// Mitsubishi GX Works2 project: LGCRFNW 23-01-2023_fr   PLC: Q06UDV

PROGRAM 00  // #1 Part Alarm
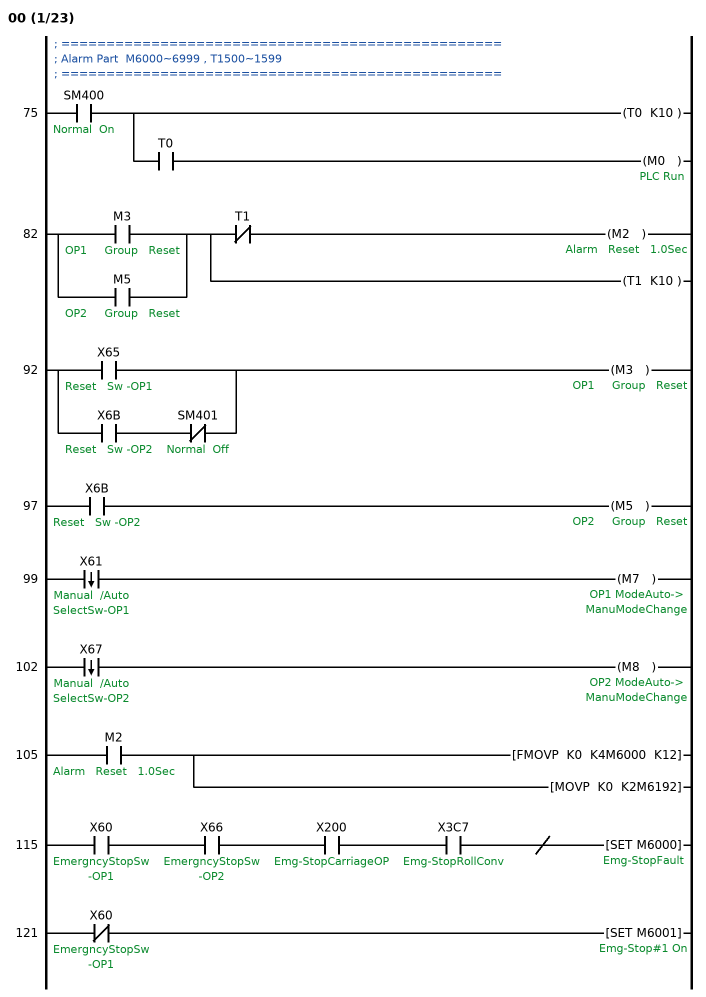
; =================================================
; Alarm Part  M6000~6999 , T1500~1599
; =================================================
75    LD      SM400  ; Normal  On
      OUT     T0 K10
      AND     T0
      OUT     M0  ; PLC Run
82    LD      M3  ; OP1     Group   Reset
      OR      M5  ; OP2     Group   Reset
      MPS
      ANI     T1
      OUT     M2  ; Alarm   Reset   1.0Sec
      MPP
      OUT     T1 K10
92    LD      X65  ; Reset   Sw -OP1
      LD      X6B  ; Reset   Sw -OP2
      ANI     SM401  ; Normal  Off
      ORB
      OUT     M3  ; OP1     Group   Reset
97    LD      X6B  ; Reset   Sw -OP2
      OUT     M5  ; OP2     Group   Reset
99    LDF     X61  ; Manual  /Auto   SelectSw-OP1
      OUT     M7  ; OP1 ModeAuto->  ManuModeChange
102   LDF     X67  ; Manual  /Auto   SelectSw-OP2
      OUT     M8  ; OP2 ModeAuto->  ManuModeChange
105   LD      M2  ; Alarm   Reset   1.0Sec
      FMOVP   K0 K4M6000 K12  ; Emg-StopFault
      MOVP    K0 K2M6192
115   LD      X60  ; EmergncyStopSw  -OP1
      AND     X66  ; EmergncyStopSw  -OP2
      AND     X200  ; Emg-StopCarriageOP
      AND     X3C7  ; Emg-StopRollConv
      INV
      SET     M6000  ; Emg-StopFault
121   LDI     X60  ; EmergncyStopSw  -OP1
      SET     M6001  ; Emg-Stop#1 On
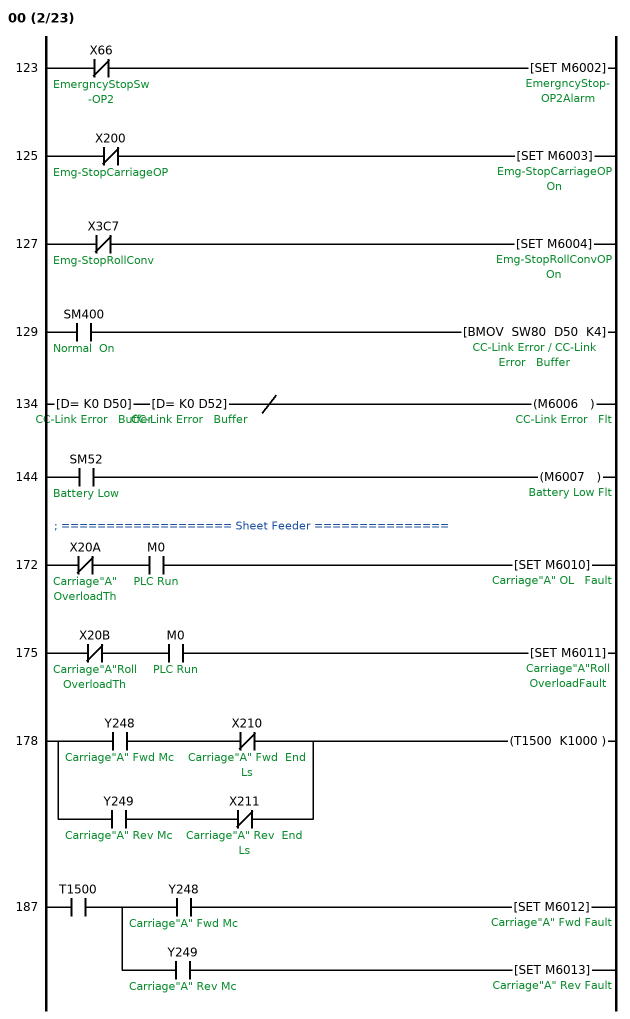
123   LDI     X66  ; EmergncyStopSw  -OP2
      SET     M6002  ; EmergncyStop-OP2Alarm
125   LDI     X200  ; Emg-StopCarriageOP
      SET     M6003  ; Emg-StopCarriageOP On
127   LDI     X3C7  ; Emg-StopRollConv
      SET     M6004  ; Emg-StopRollConvOP On
129   LD      SM400  ; Normal  On
      BMOV    SW80 D50 K4  ; CC-Link Error / CC-Link Error   Buffer
134   LDD=    K0 D50  ; CC-Link Error   Buffer
      ANDD=   K0 D52  ; CC-Link Error   Buffer
      INV
      OUT     M6006  ; CC-Link Error   Flt
144   LD      SM52  ; Battery Low
      OUT     M6007  ; Battery Low Flt
; =================== Sheet Feeder ===============
172   LDI     X20A  ; Carriage"A"     OverloadTh
      AND     M0  ; PLC Run
      SET     M6010  ; Carriage"A" OL   Fault
175   LDI     X20B  ; Carriage"A"Roll OverloadTh
      AND     M0  ; PLC Run
      SET     M6011  ; Carriage"A"Roll OverloadFault
178   LD      Y248  ; Carriage"A" Fwd Mc
      ANI     X210  ; Carriage"A" Fwd  End Ls
      LD      Y249  ; Carriage"A" Rev Mc
      ANI     X211  ; Carriage"A" Rev  End Ls
      ORB
      OUT     T1500 K1000
187   LD      T1500
      MPS
      AND     Y248  ; Carriage"A" Fwd Mc
      SET     M6012  ; Carriage"A" Fwd Fault
      MPP
      AND     Y249  ; Carriage"A" Rev Mc
      SET     M6013  ; Carriage"A" Rev Fault
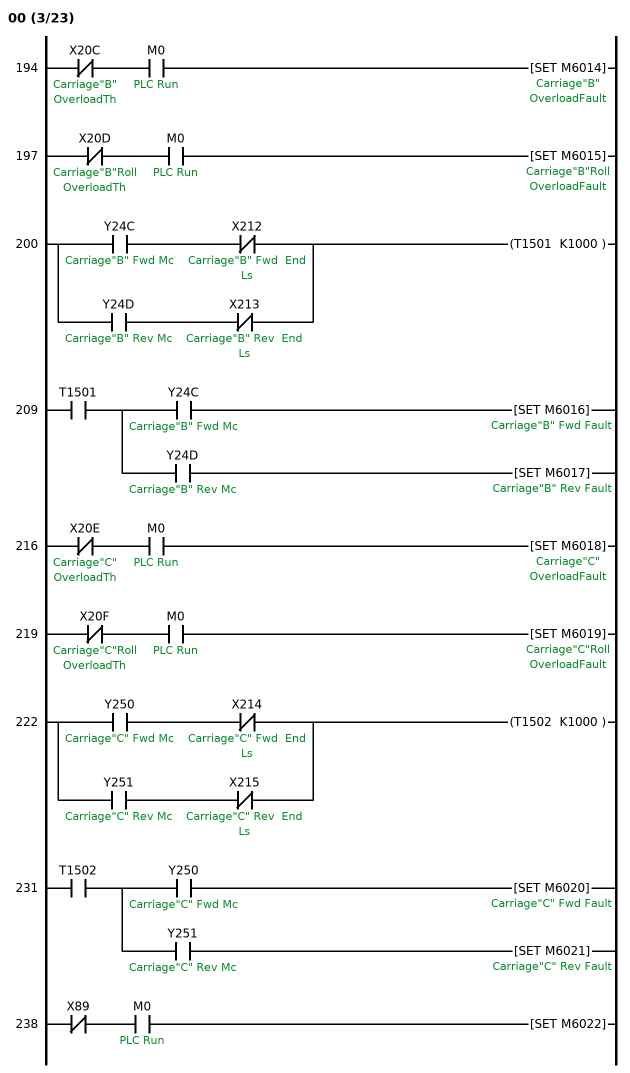
194   LDI     X20C  ; Carriage"B"     OverloadTh
      AND     M0  ; PLC Run
      SET     M6014  ; Carriage"B"     OverloadFault
197   LDI     X20D  ; Carriage"B"Roll OverloadTh
      AND     M0  ; PLC Run
      SET     M6015  ; Carriage"B"Roll OverloadFault
200   LD      Y24C  ; Carriage"B" Fwd Mc
      ANI     X212  ; Carriage"B" Fwd  End Ls
      LD      Y24D  ; Carriage"B" Rev Mc
      ANI     X213  ; Carriage"B" Rev  End Ls
      ORB
      OUT     T1501 K1000
209   LD      T1501
      MPS
      AND     Y24C  ; Carriage"B" Fwd Mc
      SET     M6016  ; Carriage"B" Fwd Fault
      MPP
      AND     Y24D  ; Carriage"B" Rev Mc
      SET     M6017  ; Carriage"B" Rev Fault
216   LDI     X20E  ; Carriage"C"     OverloadTh
      AND     M0  ; PLC Run
      SET     M6018  ; Carriage"C"     OverloadFault
219   LDI     X20F  ; Carriage"C"Roll OverloadTh
      AND     M0  ; PLC Run
      SET     M6019  ; Carriage"C"Roll OverloadFault
222   LD      Y250  ; Carriage"C" Fwd Mc
      ANI     X214  ; Carriage"C" Fwd  End Ls
      LD      Y251  ; Carriage"C" Rev Mc
      ANI     X215  ; Carriage"C" Rev  End Ls
      ORB
      OUT     T1502 K1000
231   LD      T1502
      MPS
      AND     Y250  ; Carriage"C" Fwd Mc
      SET     M6020  ; Carriage"C" Fwd Fault
      MPP
      AND     Y251  ; Carriage"C" Rev Mc
      SET     M6021  ; Carriage"C" Rev Fault
238   LDI     X89
      AND     M0  ; PLC Run
      SET     M6022
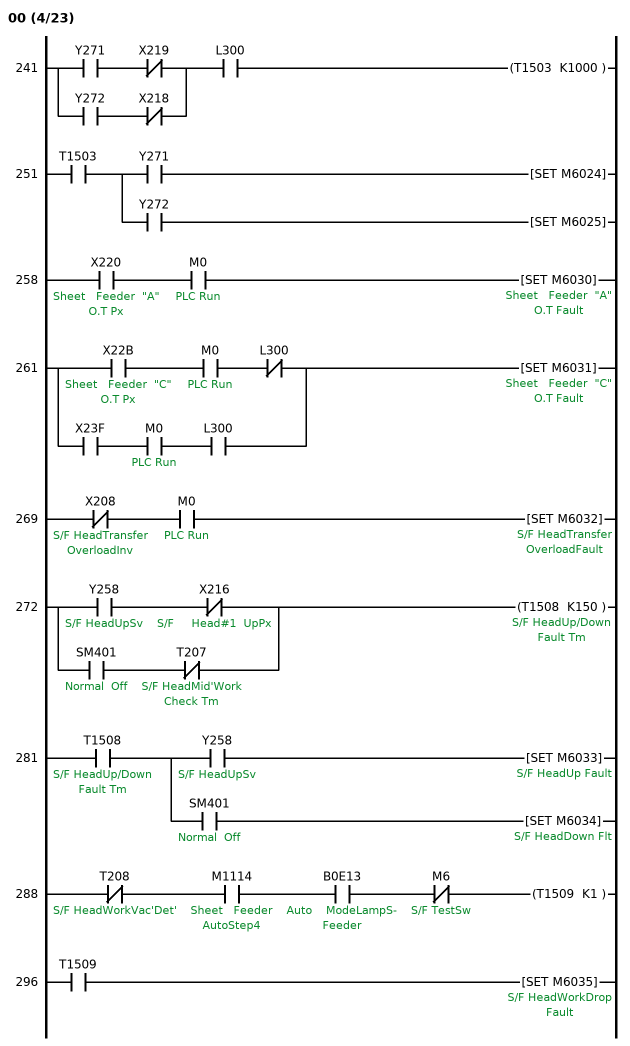
241   LD      Y271
      ANI     X219
      LD      Y272
      ANI     X218
      ORB
      AND     L300
      OUT     T1503 K1000
251   LD      T1503
      MPS
      AND     Y271
      SET     M6024
      MPP
      AND     Y272
      SET     M6025
258   LD      X220  ; Sheet   Feeder  "A" O.T Px
      AND     M0  ; PLC Run
      SET     M6030  ; Sheet   Feeder  "A" O.T Fault
261   LD      X22B  ; Sheet   Feeder  "C" O.T Px
      AND     M0  ; PLC Run
      ANI     L300
      LD      X23F
      AND     M0  ; PLC Run
      AND     L300
      ORB
      SET     M6031  ; Sheet   Feeder  "C" O.T Fault
269   LDI     X208  ; S/F HeadTransferOverloadInv
      AND     M0  ; PLC Run
      SET     M6032  ; S/F HeadTransferOverloadFault
272   LD      Y258  ; S/F HeadUpSv
      ANI     X216  ; S/F     Head#1  UpPx
      LD      SM401  ; Normal  Off
      ANI     T207  ; S/F HeadMid'WorkCheck Tm
      ORB
      OUT     T1508 K150  ; S/F HeadUp/Down Fault Tm
281   LD      T1508  ; S/F HeadUp/Down Fault Tm
      MPS
      AND     Y258  ; S/F HeadUpSv
      SET     M6033  ; S/F HeadUp Fault
      MPP
      AND     SM401  ; Normal  Off
      SET     M6034  ; S/F HeadDown Flt
288   LDI     T208  ; S/F HeadWorkVac'Det'
      AND     M1114  ; Sheet   Feeder  AutoStep4
      AND     B0E13  ; Auto    ModeLampS-Feeder
      ANI     M6  ; S/F TestSw
      OUT     T1509 K1
296   LD      T1509
      SET     M6035  ; S/F HeadWorkDropFault
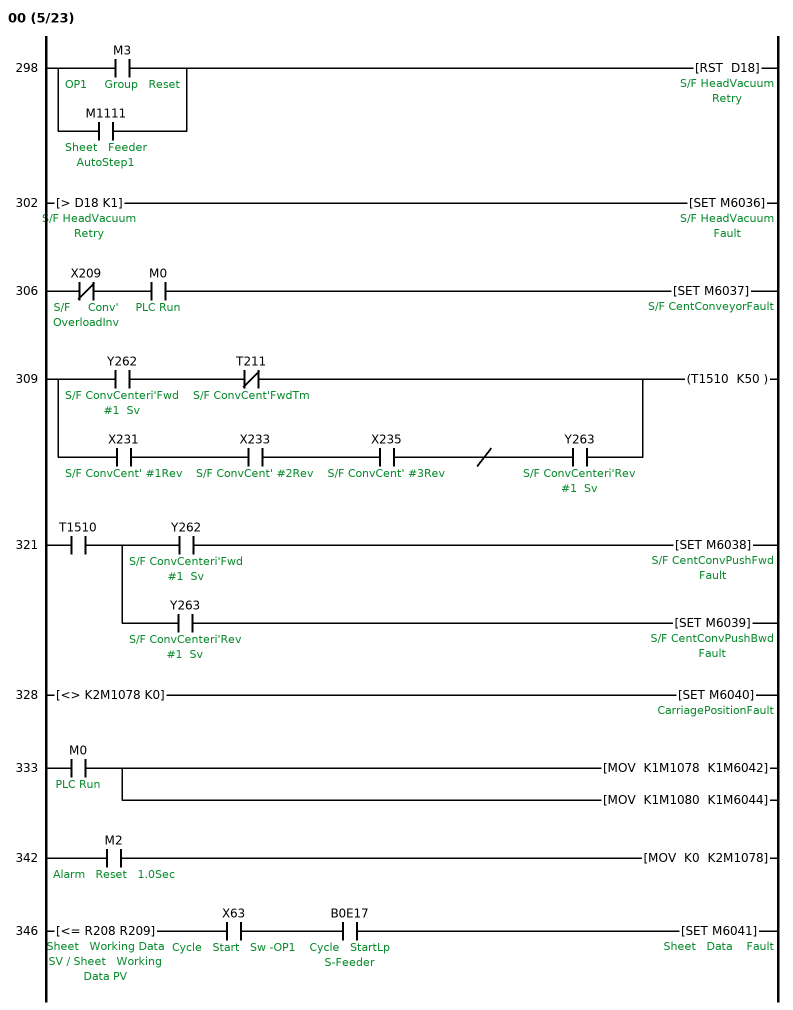
298   LD      M3  ; OP1     Group   Reset
      OR      M1111  ; Sheet   Feeder  AutoStep1
      RST     D18  ; S/F HeadVacuum  Retry
302   LD>     D18 K1  ; S/F HeadVacuum  Retry
      SET     M6036  ; S/F HeadVacuum  Fault
306   LDI     X209  ; S/F     Conv'   OverloadInv
      AND     M0  ; PLC Run
      SET     M6037  ; S/F CentConveyorFault
309   LD      Y262  ; S/F ConvCenteri'Fwd #1  Sv
      ANI     T211  ; S/F ConvCent'FwdTm
      LD      X231  ; S/F ConvCent' #1Rev
      AND     X233  ; S/F ConvCent' #2Rev
      AND     X235  ; S/F ConvCent' #3Rev
      INV
      AND     Y263  ; S/F ConvCenteri'Rev #1  Sv
      ORB
      OUT     T1510 K50
321   LD      T1510
      MPS
      AND     Y262  ; S/F ConvCenteri'Fwd #1  Sv
      SET     M6038  ; S/F CentConvPushFwdFault
      MPP
      AND     Y263  ; S/F ConvCenteri'Rev #1  Sv
      SET     M6039  ; S/F CentConvPushBwdFault
328   LD<>    K2M1078 K0  ; Carriage#1 Pos' Fault
      SET     M6040  ; CarriagePositionFault
333   LD      M0  ; PLC Run
      MOV     K1M1078 K1M6042
      MOV     K1M1080 K1M6044  ; Carriage#3 Pos'  Fault
342   LD      M2  ; Alarm   Reset   1.0Sec
      MOV     K0 K2M1078
346   LD<=    R208 R209  ; Sheet   Working Data SV / Sheet   Working Data PV
      AND     X63  ; Cycle   Start   Sw -OP1
      AND     B0E17  ; Cycle   StartLp S-Feeder
      SET     M6041  ; Sheet   Data    Fault
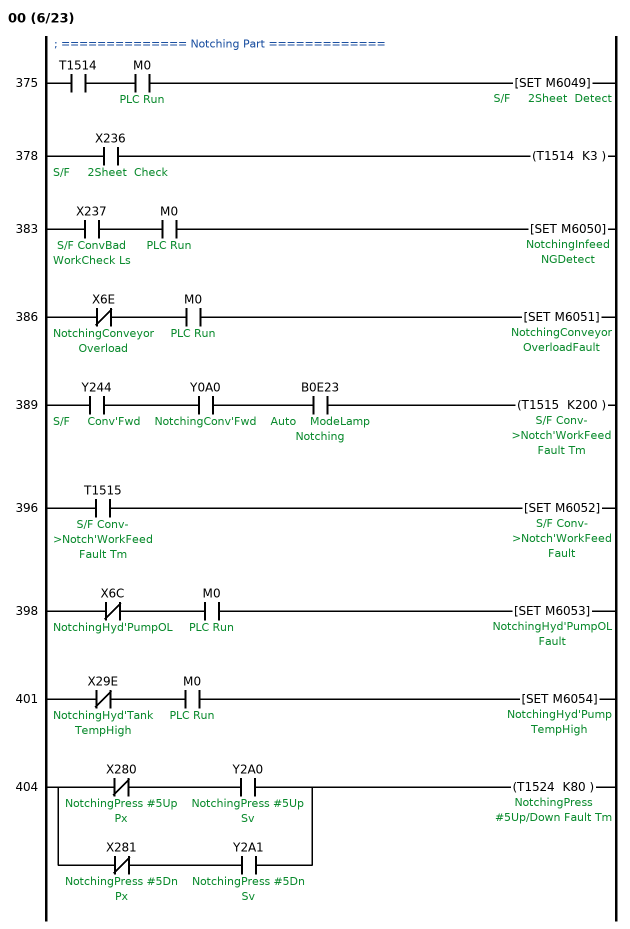
; ============== Notching Part =============
375   LD      T1514
      AND     M0  ; PLC Run
      SET     M6049  ; S/F     2Sheet  Detect
378   LD      X236  ; S/F     2Sheet  Check
      OUT     T1514 K3
383   LD      X237  ; S/F ConvBad WorkCheck Ls
      AND     M0  ; PLC Run
      SET     M6050  ; NotchingInfeedNGDetect
386   LDI     X6E  ; NotchingConveyorOverload
      AND     M0  ; PLC Run
      SET     M6051  ; NotchingConveyorOverloadFault
389   LD      Y244  ; S/F     Conv'Fwd
      AND     Y0A0  ; NotchingConv'Fwd
      AND     B0E23  ; Auto    ModeLampNotching
      OUT     T1515 K200  ; S/F Conv->Notch'WorkFeedFault Tm
396   LD      T1515  ; S/F Conv->Notch'WorkFeedFault Tm
      SET     M6052  ; S/F Conv->Notch'WorkFeedFault
398   LDI     X6C  ; NotchingHyd'PumpOL
      AND     M0  ; PLC Run
      SET     M6053  ; NotchingHyd'PumpOL Fault
401   LDI     X29E  ; NotchingHyd'TankTempHigh
      AND     M0  ; PLC Run
      SET     M6054  ; NotchingHyd'PumpTempHigh
404   LDI     X280  ; NotchingPress #5Up Px
      AND     Y2A0  ; NotchingPress #5Up Sv
      LDI     X281  ; NotchingPress #5Dn Px
      AND     Y2A1  ; NotchingPress #5Dn Sv
      ORB
      OUT     T1524 K80  ; NotchingPress #5Up/Down Fault Tm
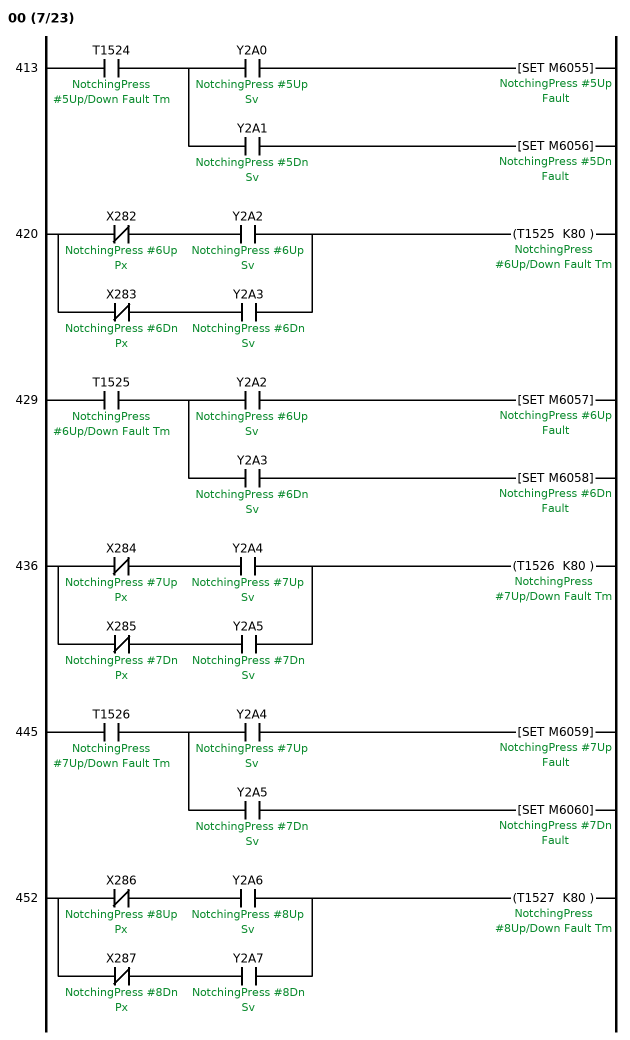
413   LD      T1524  ; NotchingPress #5Up/Down Fault Tm
      MPS
      AND     Y2A0  ; NotchingPress #5Up Sv
      SET     M6055  ; NotchingPress #5Up Fault
      MPP
      AND     Y2A1  ; NotchingPress #5Dn Sv
      SET     M6056  ; NotchingPress #5Dn Fault
420   LDI     X282  ; NotchingPress #6Up Px
      AND     Y2A2  ; NotchingPress #6Up Sv
      LDI     X283  ; NotchingPress #6Dn Px
      AND     Y2A3  ; NotchingPress #6Dn Sv
      ORB
      OUT     T1525 K80  ; NotchingPress #6Up/Down Fault Tm
429   LD      T1525  ; NotchingPress #6Up/Down Fault Tm
      MPS
      AND     Y2A2  ; NotchingPress #6Up Sv
      SET     M6057  ; NotchingPress #6Up Fault
      MPP
      AND     Y2A3  ; NotchingPress #6Dn Sv
      SET     M6058  ; NotchingPress #6Dn Fault
436   LDI     X284  ; NotchingPress #7Up Px
      AND     Y2A4  ; NotchingPress #7Up Sv
      LDI     X285  ; NotchingPress #7Dn Px
      AND     Y2A5  ; NotchingPress #7Dn Sv
      ORB
      OUT     T1526 K80  ; NotchingPress #7Up/Down Fault Tm
445   LD      T1526  ; NotchingPress #7Up/Down Fault Tm
      MPS
      AND     Y2A4  ; NotchingPress #7Up Sv
      SET     M6059  ; NotchingPress #7Up Fault
      MPP
      AND     Y2A5  ; NotchingPress #7Dn Sv
      SET     M6060  ; NotchingPress #7Dn Fault
452   LDI     X286  ; NotchingPress #8Up Px
      AND     Y2A6  ; NotchingPress #8Up Sv
      LDI     X287  ; NotchingPress #8Dn Px
      AND     Y2A7  ; NotchingPress #8Dn Sv
      ORB
      OUT     T1527 K80  ; NotchingPress #8Up/Down Fault Tm
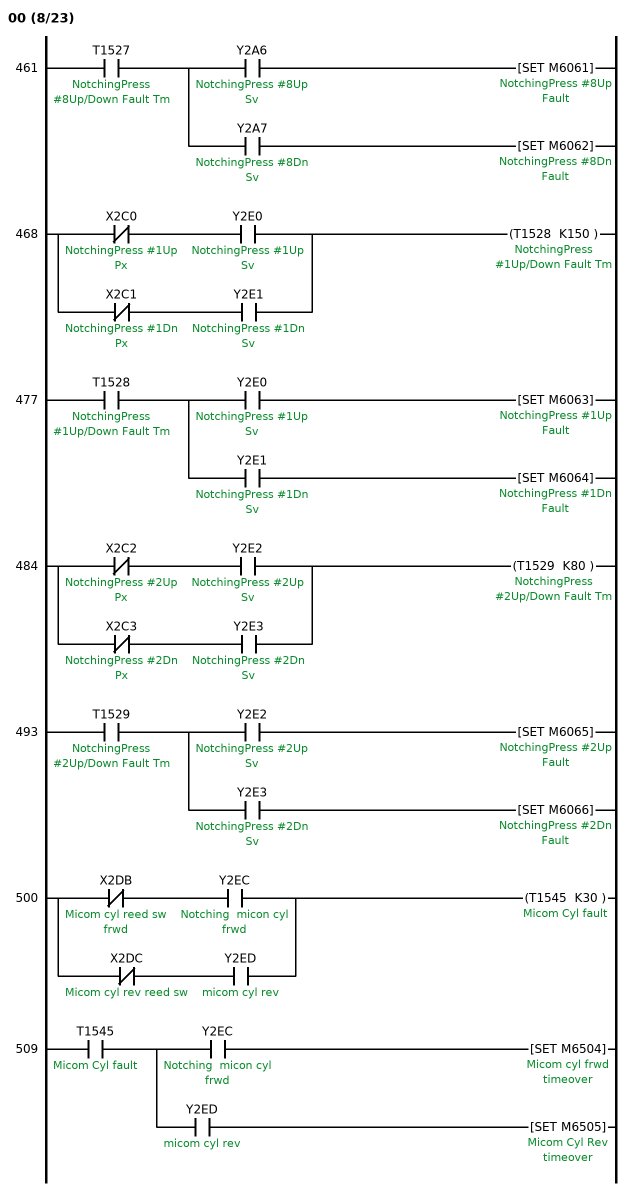
461   LD      T1527  ; NotchingPress #8Up/Down Fault Tm
      MPS
      AND     Y2A6  ; NotchingPress #8Up Sv
      SET     M6061  ; NotchingPress #8Up Fault
      MPP
      AND     Y2A7  ; NotchingPress #8Dn Sv
      SET     M6062  ; NotchingPress #8Dn Fault
468   LDI     X2C0  ; NotchingPress #1Up Px
      AND     Y2E0  ; NotchingPress #1Up Sv
      LDI     X2C1  ; NotchingPress #1Dn Px
      AND     Y2E1  ; NotchingPress #1Dn Sv
      ORB
      OUT     T1528 K150  ; NotchingPress #1Up/Down Fault Tm
477   LD      T1528  ; NotchingPress #1Up/Down Fault Tm
      MPS
      AND     Y2E0  ; NotchingPress #1Up Sv
      SET     M6063  ; NotchingPress #1Up Fault
      MPP
      AND     Y2E1  ; NotchingPress #1Dn Sv
      SET     M6064  ; NotchingPress #1Dn Fault
484   LDI     X2C2  ; NotchingPress #2Up Px
      AND     Y2E2  ; NotchingPress #2Up Sv
      LDI     X2C3  ; NotchingPress #2Dn Px
      AND     Y2E3  ; NotchingPress #2Dn Sv
      ORB
      OUT     T1529 K80  ; NotchingPress #2Up/Down Fault Tm
493   LD      T1529  ; NotchingPress #2Up/Down Fault Tm
      MPS
      AND     Y2E2  ; NotchingPress #2Up Sv
      SET     M6065  ; NotchingPress #2Up Fault
      MPP
      AND     Y2E3  ; NotchingPress #2Dn Sv
      SET     M6066  ; NotchingPress #2Dn Fault
500   LDI     X2DB  ; Micom cyl reed sw frwd
      AND     Y2EC  ; Notching  micon cyl frwd
      LDI     X2DC  ; Micom cyl rev reed sw
      AND     Y2ED  ; micom cyl rev
      ORB
      OUT     T1545 K30  ; Micom Cyl fault
509   LD      T1545  ; Micom Cyl fault
      MPS
      AND     Y2EC  ; Notching  micon cyl frwd
      SET     M6504  ; Micom cyl frwd timeover
      MPP
      AND     Y2ED  ; micom cyl rev
      SET     M6505  ; Micom Cyl Rev timeover
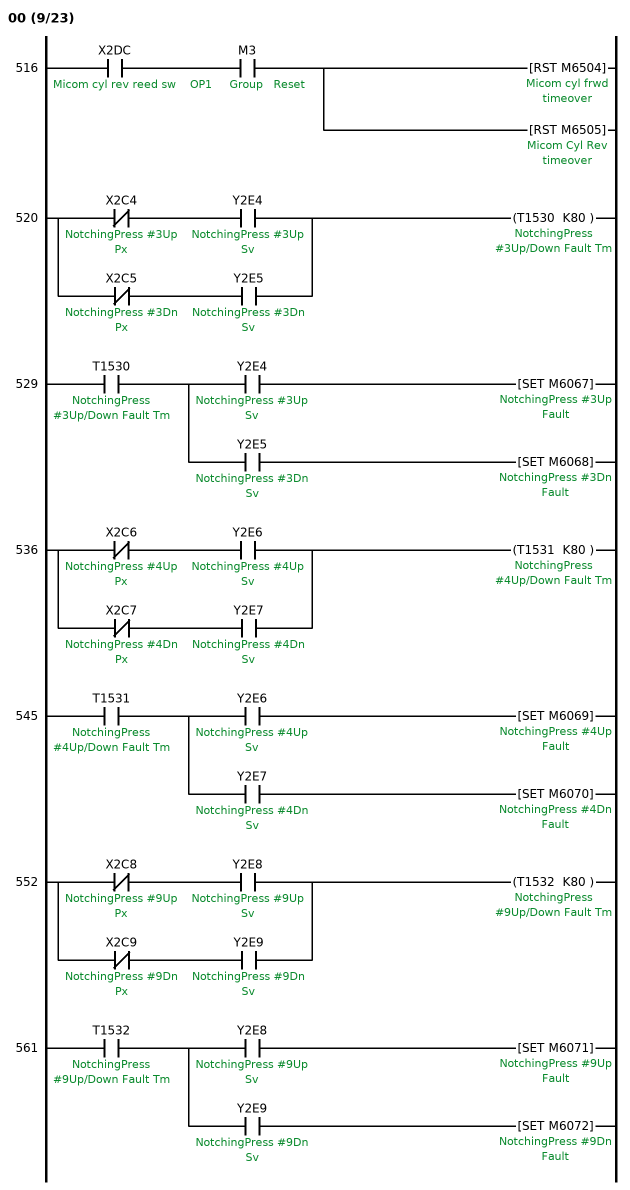
516   LD      X2DC  ; Micom cyl rev reed sw
      AND     M3  ; OP1     Group   Reset
      RST     M6504  ; Micom cyl frwd timeover
      RST     M6505  ; Micom Cyl Rev timeover
520   LDI     X2C4  ; NotchingPress #3Up Px
      AND     Y2E4  ; NotchingPress #3Up Sv
      LDI     X2C5  ; NotchingPress #3Dn Px
      AND     Y2E5  ; NotchingPress #3Dn Sv
      ORB
      OUT     T1530 K80  ; NotchingPress #3Up/Down Fault Tm
529   LD      T1530  ; NotchingPress #3Up/Down Fault Tm
      MPS
      AND     Y2E4  ; NotchingPress #3Up Sv
      SET     M6067  ; NotchingPress #3Up Fault
      MPP
      AND     Y2E5  ; NotchingPress #3Dn Sv
      SET     M6068  ; NotchingPress #3Dn Fault
536   LDI     X2C6  ; NotchingPress #4Up Px
      AND     Y2E6  ; NotchingPress #4Up Sv
      LDI     X2C7  ; NotchingPress #4Dn Px
      AND     Y2E7  ; NotchingPress #4Dn Sv
      ORB
      OUT     T1531 K80  ; NotchingPress #4Up/Down Fault Tm
545   LD      T1531  ; NotchingPress #4Up/Down Fault Tm
      MPS
      AND     Y2E6  ; NotchingPress #4Up Sv
      SET     M6069  ; NotchingPress #4Up Fault
      MPP
      AND     Y2E7  ; NotchingPress #4Dn Sv
      SET     M6070  ; NotchingPress #4Dn Fault
552   LDI     X2C8  ; NotchingPress #9Up Px
      AND     Y2E8  ; NotchingPress #9Up Sv
      LDI     X2C9  ; NotchingPress #9Dn Px
      AND     Y2E9  ; NotchingPress #9Dn Sv
      ORB
      OUT     T1532 K80  ; NotchingPress #9Up/Down Fault Tm
561   LD      T1532  ; NotchingPress #9Up/Down Fault Tm
      MPS
      AND     Y2E8  ; NotchingPress #9Up Sv
      SET     M6071  ; NotchingPress #9Up Fault
      MPP
      AND     Y2E9  ; NotchingPress #9Dn Sv
      SET     M6072  ; NotchingPress #9Dn Fault
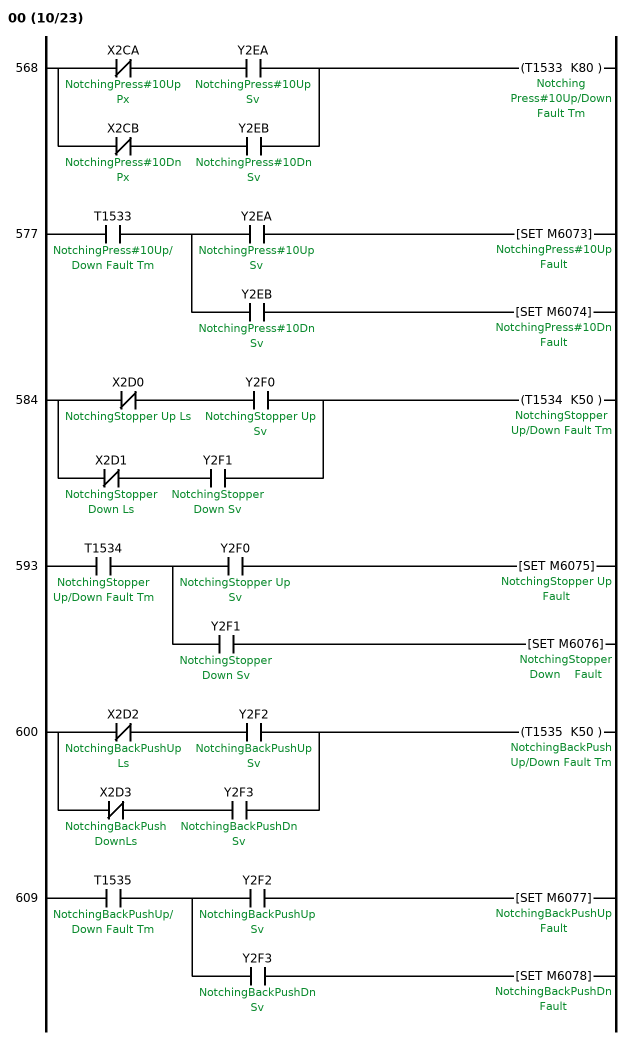
568   LDI     X2CA  ; NotchingPress#10Up Px
      AND     Y2EA  ; NotchingPress#10Up Sv
      LDI     X2CB  ; NotchingPress#10Dn Px
      AND     Y2EB  ; NotchingPress#10Dn Sv
      ORB
      OUT     T1533 K80  ; NotchingPress#10Up/Down Fault Tm
577   LD      T1533  ; NotchingPress#10Up/Down Fault Tm
      MPS
      AND     Y2EA  ; NotchingPress#10Up Sv
      SET     M6073  ; NotchingPress#10Up Fault
      MPP
      AND     Y2EB  ; NotchingPress#10Dn Sv
      SET     M6074  ; NotchingPress#10Dn Fault
584   LDI     X2D0  ; NotchingStopper Up Ls
      AND     Y2F0  ; NotchingStopper Up Sv
      LDI     X2D1  ; NotchingStopper Down Ls
      AND     Y2F1  ; NotchingStopper Down Sv
      ORB
      OUT     T1534 K50  ; NotchingStopper Up/Down Fault Tm
593   LD      T1534  ; NotchingStopper Up/Down Fault Tm
      MPS
      AND     Y2F0  ; NotchingStopper Up Sv
      SET     M6075  ; NotchingStopper Up Fault
      MPP
      AND     Y2F1  ; NotchingStopper Down Sv
      SET     M6076  ; NotchingStopper Down    Fault
600   LDI     X2D2  ; NotchingBackPushUpLs
      AND     Y2F2  ; NotchingBackPushUpSv
      LDI     X2D3  ; NotchingBackPushDownLs
      AND     Y2F3  ; NotchingBackPushDnSv
      ORB
      OUT     T1535 K50  ; NotchingBackPushUp/Down Fault Tm
609   LD      T1535  ; NotchingBackPushUp/Down Fault Tm
      MPS
      AND     Y2F2  ; NotchingBackPushUpSv
      SET     M6077  ; NotchingBackPushUpFault
      MPP
      AND     Y2F3  ; NotchingBackPushDnSv
      SET     M6078  ; NotchingBackPushDnFault
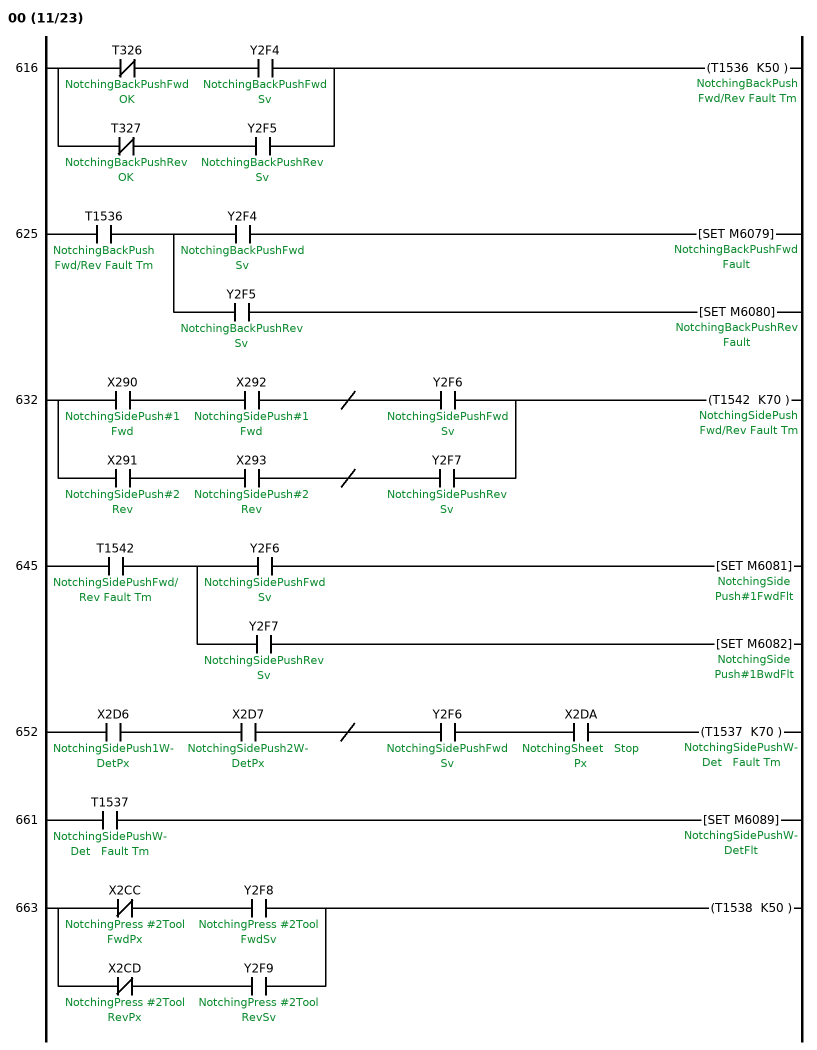
616   LDI     T326  ; NotchingBackPushFwd OK
      AND     Y2F4  ; NotchingBackPushFwdSv
      LDI     T327  ; NotchingBackPushRev OK
      AND     Y2F5  ; NotchingBackPushRevSv
      ORB
      OUT     T1536 K50  ; NotchingBackPushFwd/Rev Fault Tm
625   LD      T1536  ; NotchingBackPushFwd/Rev Fault Tm
      MPS
      AND     Y2F4  ; NotchingBackPushFwdSv
      SET     M6079  ; NotchingBackPushFwdFault
      MPP
      AND     Y2F5  ; NotchingBackPushRevSv
      SET     M6080  ; NotchingBackPushRevFault
632   LD      X290  ; NotchingSidePush#1 Fwd
      AND     X292  ; NotchingSidePush#1 Fwd
      INV
      AND     Y2F6  ; NotchingSidePushFwd Sv
      LD      X291  ; NotchingSidePush#2 Rev
      AND     X293  ; NotchingSidePush#2 Rev
      INV
      AND     Y2F7  ; NotchingSidePushRev Sv
      ORB
      OUT     T1542 K70  ; NotchingSidePushFwd/Rev Fault Tm
645   LD      T1542  ; NotchingSidePushFwd/Rev Fault Tm
      MPS
      AND     Y2F6  ; NotchingSidePushFwd Sv
      SET     M6081  ; NotchingSidePush#1FwdFlt
      MPP
      AND     Y2F7  ; NotchingSidePushRev Sv
      SET     M6082  ; NotchingSidePush#1BwdFlt
652   LD      X2D6  ; NotchingSidePush1W-DetPx
      AND     X2D7  ; NotchingSidePush2W-DetPx
      INV
      AND     Y2F6  ; NotchingSidePushFwd Sv
      AND     X2DA  ; NotchingSheet   Stop Px
      OUT     T1537 K70  ; NotchingSidePushW-Det   Fault Tm
661   LD      T1537  ; NotchingSidePushW-Det   Fault Tm
      SET     M6089  ; NotchingSidePushW-DetFlt
663   LDI     X2CC  ; NotchingPress #2Tool FwdPx
      AND     Y2F8  ; NotchingPress #2Tool FwdSv
      LDI     X2CD  ; NotchingPress #2Tool RevPx
      AND     Y2F9  ; NotchingPress #2Tool RevSv
      ORB
      OUT     T1538 K50
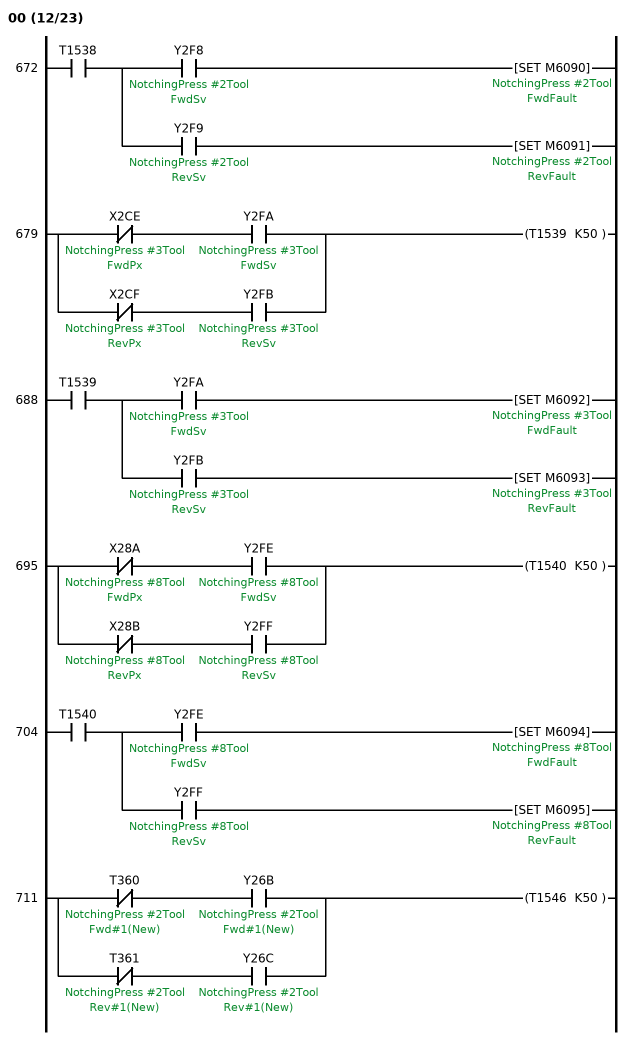
672   LD      T1538
      MPS
      AND     Y2F8  ; NotchingPress #2Tool FwdSv
      SET     M6090  ; NotchingPress #2Tool FwdFault
      MPP
      AND     Y2F9  ; NotchingPress #2Tool RevSv
      SET     M6091  ; NotchingPress #2Tool RevFault
679   LDI     X2CE  ; NotchingPress #3Tool FwdPx
      AND     Y2FA  ; NotchingPress #3Tool FwdSv
      LDI     X2CF  ; NotchingPress #3Tool RevPx
      AND     Y2FB  ; NotchingPress #3Tool RevSv
      ORB
      OUT     T1539 K50
688   LD      T1539
      MPS
      AND     Y2FA  ; NotchingPress #3Tool FwdSv
      SET     M6092  ; NotchingPress #3Tool FwdFault
      MPP
      AND     Y2FB  ; NotchingPress #3Tool RevSv
      SET     M6093  ; NotchingPress #3Tool RevFault
695   LDI     X28A  ; NotchingPress #8Tool FwdPx
      AND     Y2FE  ; NotchingPress #8Tool FwdSv
      LDI     X28B  ; NotchingPress #8Tool RevPx
      AND     Y2FF  ; NotchingPress #8Tool RevSv
      ORB
      OUT     T1540 K50
704   LD      T1540
      MPS
      AND     Y2FE  ; NotchingPress #8Tool FwdSv
      SET     M6094  ; NotchingPress #8Tool FwdFault
      MPP
      AND     Y2FF  ; NotchingPress #8Tool RevSv
      SET     M6095  ; NotchingPress #8Tool RevFault
711   LDI     T360  ; NotchingPress #2Tool Fwd#1(New)
      AND     Y26B  ; NotchingPress #2Tool Fwd#1(New)
      LDI     T361  ; NotchingPress #2Tool Rev#1(New)
      AND     Y26C  ; NotchingPress #2Tool Rev#1(New)
      ORB
      OUT     T1546 K50
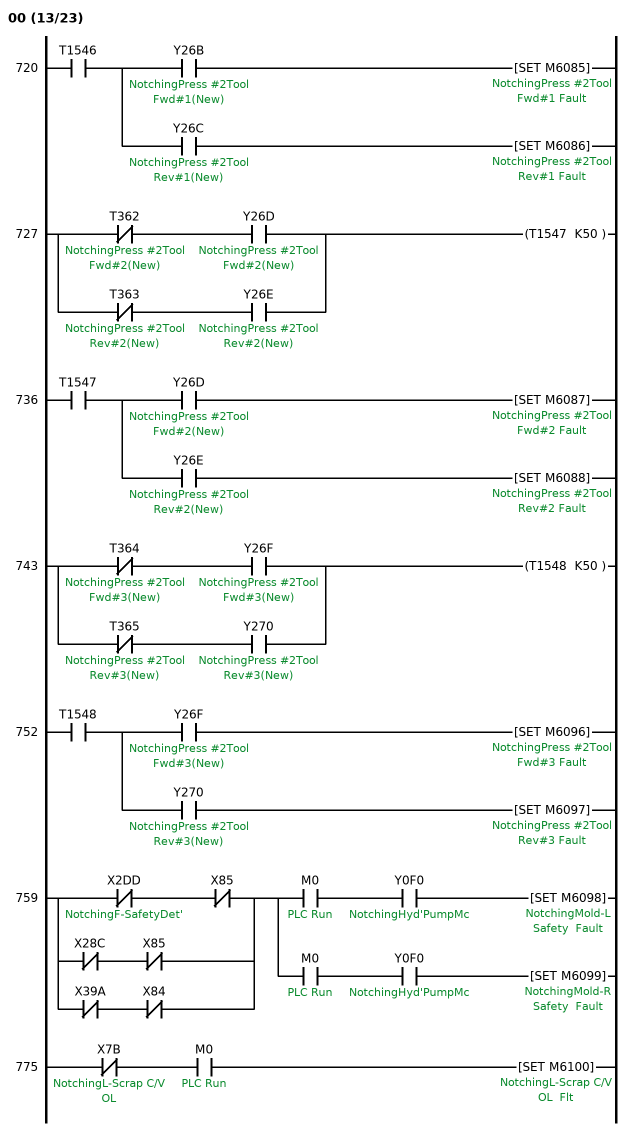
720   LD      T1546
      MPS
      AND     Y26B  ; NotchingPress #2Tool Fwd#1(New)
      SET     M6085  ; NotchingPress #2Tool Fwd#1 Fault
      MPP
      AND     Y26C  ; NotchingPress #2Tool Rev#1(New)
      SET     M6086  ; NotchingPress #2Tool Rev#1 Fault
727   LDI     T362  ; NotchingPress #2Tool Fwd#2(New)
      AND     Y26D  ; NotchingPress #2Tool Fwd#2(New)
      LDI     T363  ; NotchingPress #2Tool Rev#2(New)
      AND     Y26E  ; NotchingPress #2Tool Rev#2(New)
      ORB
      OUT     T1547 K50
736   LD      T1547
      MPS
      AND     Y26D  ; NotchingPress #2Tool Fwd#2(New)
      SET     M6087  ; NotchingPress #2Tool Fwd#2 Fault
      MPP
      AND     Y26E  ; NotchingPress #2Tool Rev#2(New)
      SET     M6088  ; NotchingPress #2Tool Rev#2 Fault
743   LDI     T364  ; NotchingPress #2Tool Fwd#3(New)
      AND     Y26F  ; NotchingPress #2Tool Fwd#3(New)
      LDI     T365  ; NotchingPress #2Tool Rev#3(New)
      AND     Y270  ; NotchingPress #2Tool Rev#3(New)
      ORB
      OUT     T1548 K50
752   LD      T1548
      MPS
      AND     Y26F  ; NotchingPress #2Tool Fwd#3(New)
      SET     M6096  ; NotchingPress #2Tool Fwd#3 Fault
      MPP
      AND     Y270  ; NotchingPress #2Tool Rev#3(New)
      SET     M6097  ; NotchingPress #2Tool Rev#3 Fault
759   LDI     X2DD  ; NotchingF-SafetyDet'
      ANI     X85
      LDI     X28C
      ANI     X85
      ORB
      LDI     X39A
      ANI     X84
      ORB
      MPS
      AND     M0  ; PLC Run
      AND     Y0F0  ; NotchingHyd'PumpMc
      SET     M6098  ; NotchingMold-L  Safety  Fault
      MPP
      AND     M0  ; PLC Run
      AND     Y0F0  ; NotchingHyd'PumpMc
      SET     M6099  ; NotchingMold-R  Safety  Fault
775   LDI     X7B  ; NotchingL-Scrap C/V OL
      AND     M0  ; PLC Run
      SET     M6100  ; NotchingL-Scrap C/V OL  Flt
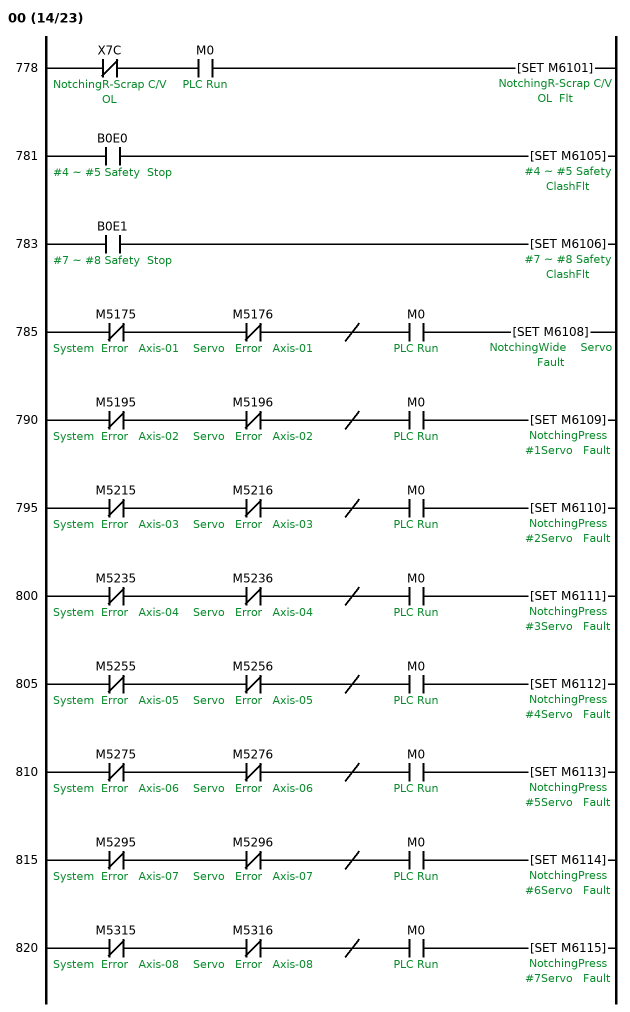
778   LDI     X7C  ; NotchingR-Scrap C/V OL
      AND     M0  ; PLC Run
      SET     M6101  ; NotchingR-Scrap C/V OL  Flt
781   LD      B0E0  ; #4 ~ #5 Safety  Stop
      SET     M6105  ; #4 ~ #5 Safety  ClashFlt
783   LD      B0E1  ; #7 ~ #8 Safety  Stop
      SET     M6106  ; #7 ~ #8 Safety  ClashFlt
785   LDI     M5175  ; System  Error   Axis-01
      ANI     M5176  ; Servo   Error   Axis-01
      INV
      AND     M0  ; PLC Run
      SET     M6108  ; NotchingWide    Servo   Fault
790   LDI     M5195  ; System  Error   Axis-02
      ANI     M5196  ; Servo   Error   Axis-02
      INV
      AND     M0  ; PLC Run
      SET     M6109  ; NotchingPress #1Servo   Fault
795   LDI     M5215  ; System  Error   Axis-03
      ANI     M5216  ; Servo   Error   Axis-03
      INV
      AND     M0  ; PLC Run
      SET     M6110  ; NotchingPress #2Servo   Fault
800   LDI     M5235  ; System  Error   Axis-04
      ANI     M5236  ; Servo   Error   Axis-04
      INV
      AND     M0  ; PLC Run
      SET     M6111  ; NotchingPress #3Servo   Fault
805   LDI     M5255  ; System  Error   Axis-05
      ANI     M5256  ; Servo   Error   Axis-05
      INV
      AND     M0  ; PLC Run
      SET     M6112  ; NotchingPress #4Servo   Fault
810   LDI     M5275  ; System  Error   Axis-06
      ANI     M5276  ; Servo   Error   Axis-06
      INV
      AND     M0  ; PLC Run
      SET     M6113  ; NotchingPress #5Servo   Fault
815   LDI     M5295  ; System  Error   Axis-07
      ANI     M5296  ; Servo   Error   Axis-07
      INV
      AND     M0  ; PLC Run
      SET     M6114  ; NotchingPress #6Servo   Fault
820   LDI     M5315  ; System  Error   Axis-08
      ANI     M5316  ; Servo   Error   Axis-08
      INV
      AND     M0  ; PLC Run
      SET     M6115  ; NotchingPress #7Servo   Fault
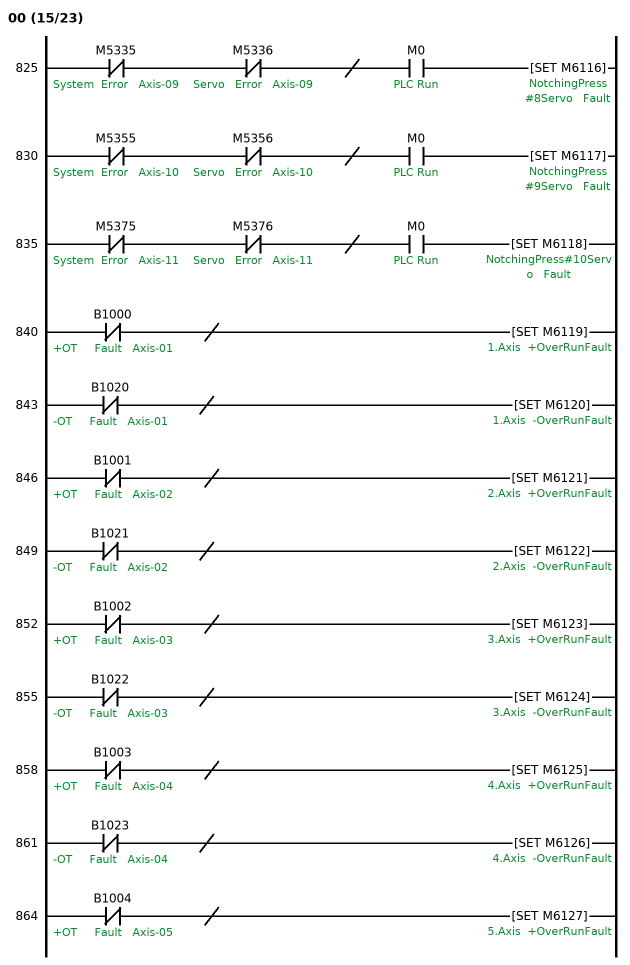
825   LDI     M5335  ; System  Error   Axis-09
      ANI     M5336  ; Servo   Error   Axis-09
      INV
      AND     M0  ; PLC Run
      SET     M6116  ; NotchingPress #8Servo   Fault
830   LDI     M5355  ; System  Error   Axis-10
      ANI     M5356  ; Servo   Error   Axis-10
      INV
      AND     M0  ; PLC Run
      SET     M6117  ; NotchingPress #9Servo   Fault
835   LDI     M5375  ; System  Error   Axis-11
      ANI     M5376  ; Servo   Error   Axis-11
      INV
      AND     M0  ; PLC Run
      SET     M6118  ; NotchingPress#10Servo   Fault
840   LDI     B1000  ; +OT     Fault   Axis-01
      INV
      SET     M6119  ; 1.Axis  +OverRunFault
843   LDI     B1020  ; -OT     Fault   Axis-01
      INV
      SET     M6120  ; 1.Axis  -OverRunFault
846   LDI     B1001  ; +OT     Fault   Axis-02
      INV
      SET     M6121  ; 2.Axis  +OverRunFault
849   LDI     B1021  ; -OT     Fault   Axis-02
      INV
      SET     M6122  ; 2.Axis  -OverRunFault
852   LDI     B1002  ; +OT     Fault   Axis-03
      INV
      SET     M6123  ; 3.Axis  +OverRunFault
855   LDI     B1022  ; -OT     Fault   Axis-03
      INV
      SET     M6124  ; 3.Axis  -OverRunFault
858   LDI     B1003  ; +OT     Fault   Axis-04
      INV
      SET     M6125  ; 4.Axis  +OverRunFault
861   LDI     B1023  ; -OT     Fault   Axis-04
      INV
      SET     M6126  ; 4.Axis  -OverRunFault
864   LDI     B1004  ; +OT     Fault   Axis-05
      INV
      SET     M6127  ; 5.Axis  +OverRunFault
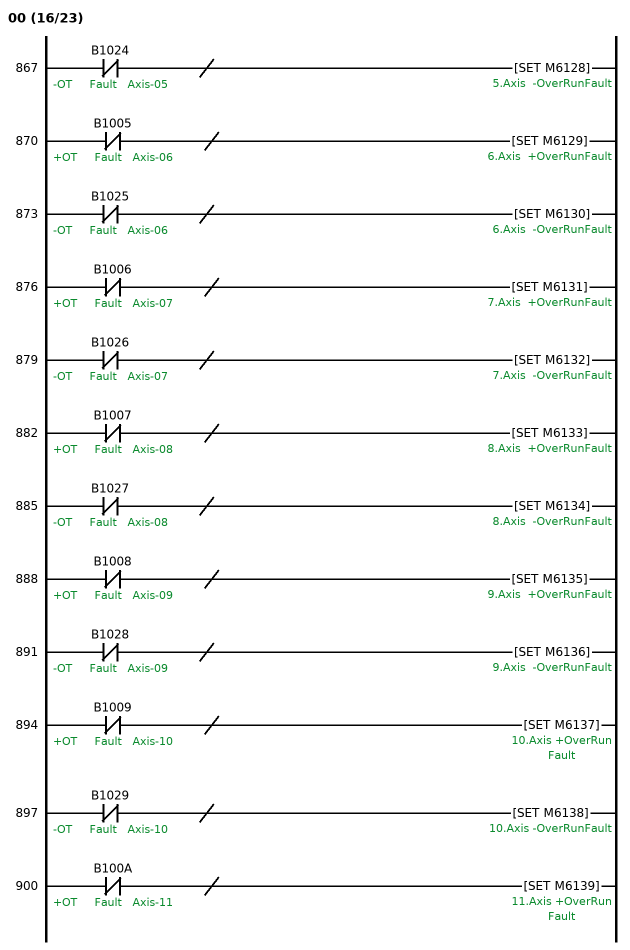
867   LDI     B1024  ; -OT     Fault   Axis-05
      INV
      SET     M6128  ; 5.Axis  -OverRunFault
870   LDI     B1005  ; +OT     Fault   Axis-06
      INV
      SET     M6129  ; 6.Axis  +OverRunFault
873   LDI     B1025  ; -OT     Fault   Axis-06
      INV
      SET     M6130  ; 6.Axis  -OverRunFault
876   LDI     B1006  ; +OT     Fault   Axis-07
      INV
      SET     M6131  ; 7.Axis  +OverRunFault
879   LDI     B1026  ; -OT     Fault   Axis-07
      INV
      SET     M6132  ; 7.Axis  -OverRunFault
882   LDI     B1007  ; +OT     Fault   Axis-08
      INV
      SET     M6133  ; 8.Axis  +OverRunFault
885   LDI     B1027  ; -OT     Fault   Axis-08
      INV
      SET     M6134  ; 8.Axis  -OverRunFault
888   LDI     B1008  ; +OT     Fault   Axis-09
      INV
      SET     M6135  ; 9.Axis  +OverRunFault
891   LDI     B1028  ; -OT     Fault   Axis-09
      INV
      SET     M6136  ; 9.Axis  -OverRunFault
894   LDI     B1009  ; +OT     Fault   Axis-10
      INV
      SET     M6137  ; 10.Axis +OverRunFault
897   LDI     B1029  ; -OT     Fault   Axis-10
      INV
      SET     M6138  ; 10.Axis -OverRunFault
900   LDI     B100A  ; +OT     Fault   Axis-11
      INV
      SET     M6139  ; 11.Axis +OverRunFault
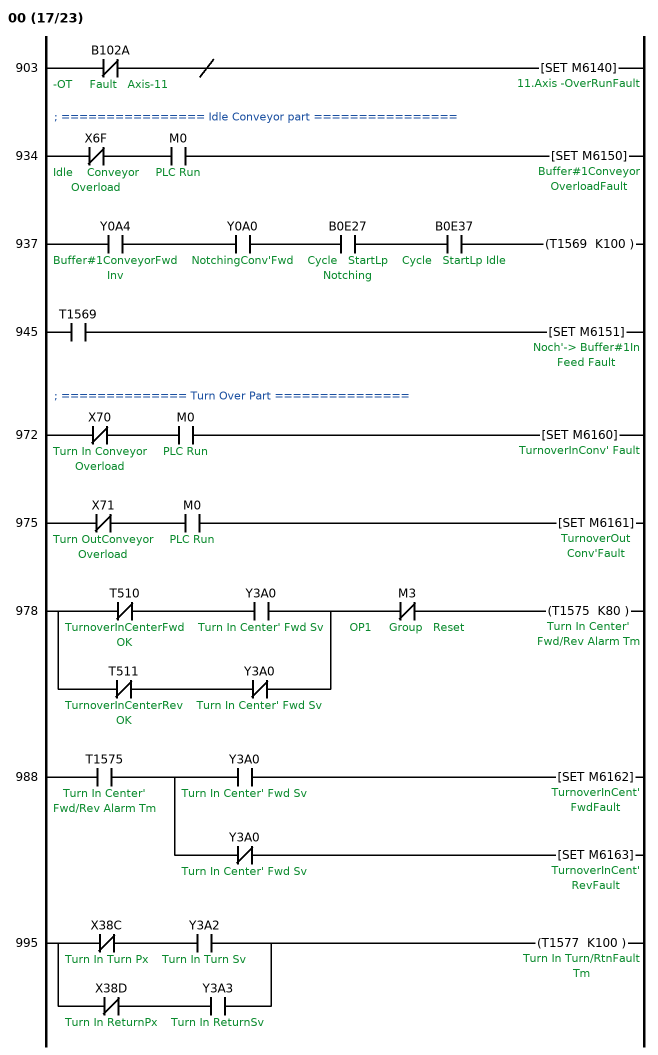
903   LDI     B102A  ; -OT     Fault   Axis-11
      INV
      SET     M6140  ; 11.Axis -OverRunFault
; ================ Idle Conveyor part ================
934   LDI     X6F  ; Idle    ConveyorOverload
      AND     M0  ; PLC Run
      SET     M6150  ; Buffer#1ConveyorOverloadFault
937   LD      Y0A4  ; Buffer#1ConveyorFwd Inv
      AND     Y0A0  ; NotchingConv'Fwd
      AND     B0E27  ; Cycle   StartLp Notching
      AND     B0E37  ; Cycle   StartLp Idle
      OUT     T1569 K100
945   LD      T1569
      SET     M6151  ; Noch'-> Buffer#1In Feed Fault
; ============== Turn Over Part ===============
972   LDI     X70  ; Turn In ConveyorOverload
      AND     M0  ; PLC Run
      SET     M6160  ; TurnoverInConv' Fault
975   LDI     X71  ; Turn OutConveyorOverload
      AND     M0  ; PLC Run
      SET     M6161  ; TurnoverOutConv'Fault
978   LDI     T510  ; TurnoverInCenterFwd OK
      AND     Y3A0  ; Turn In Center' Fwd Sv
      LDI     T511  ; TurnoverInCenterRev OK
      ANI     Y3A0  ; Turn In Center' Fwd Sv
      ORB
      ANI     M3  ; OP1     Group   Reset
      OUT     T1575 K80  ; Turn In Center' Fwd/Rev Alarm Tm
988   LD      T1575  ; Turn In Center' Fwd/Rev Alarm Tm
      MPS
      AND     Y3A0  ; Turn In Center' Fwd Sv
      SET     M6162  ; TurnoverInCent' FwdFault
      MPP
      ANI     Y3A0  ; Turn In Center' Fwd Sv
      SET     M6163  ; TurnoverInCent' RevFault
995   LDI     X38C  ; Turn In Turn Px
      AND     Y3A2  ; Turn In Turn Sv
      LDI     X38D  ; Turn In ReturnPx
      AND     Y3A3  ; Turn In ReturnSv
      ORB
      OUT     T1577 K100  ; Turn In Turn/RtnFault Tm
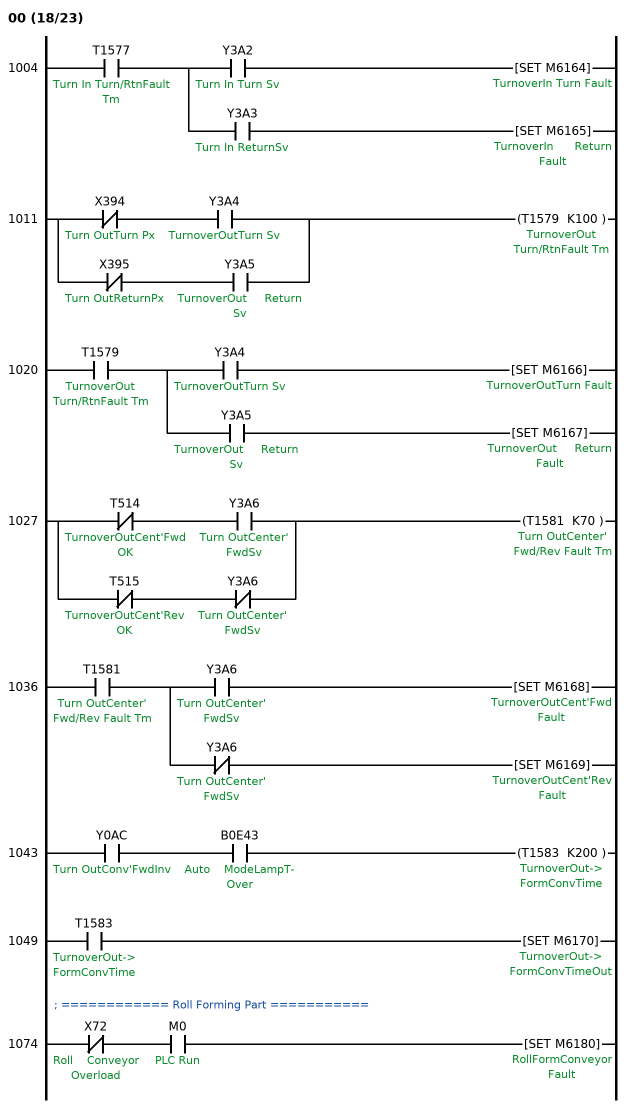
1004  LD      T1577  ; Turn In Turn/RtnFault Tm
      MPS
      AND     Y3A2  ; Turn In Turn Sv
      SET     M6164  ; TurnoverIn Turn Fault
      MPP
      AND     Y3A3  ; Turn In ReturnSv
      SET     M6165  ; TurnoverIn      Return  Fault
1011  LDI     X394  ; Turn OutTurn Px
      AND     Y3A4  ; TurnoverOutTurn Sv
      LDI     X395  ; Turn OutReturnPx
      AND     Y3A5  ; TurnoverOut     Return  Sv
      ORB
      OUT     T1579 K100  ; TurnoverOut     Turn/RtnFault Tm
1020  LD      T1579  ; TurnoverOut     Turn/RtnFault Tm
      MPS
      AND     Y3A4  ; TurnoverOutTurn Sv
      SET     M6166  ; TurnoverOutTurn Fault
      MPP
      AND     Y3A5  ; TurnoverOut     Return  Sv
      SET     M6167  ; TurnoverOut     Return  Fault
1027  LDI     T514  ; TurnoverOutCent'Fwd OK
      AND     Y3A6  ; Turn OutCenter' FwdSv
      LDI     T515  ; TurnoverOutCent'Rev OK
      ANI     Y3A6  ; Turn OutCenter' FwdSv
      ORB
      OUT     T1581 K70  ; Turn OutCenter' Fwd/Rev Fault Tm
1036  LD      T1581  ; Turn OutCenter' Fwd/Rev Fault Tm
      MPS
      AND     Y3A6  ; Turn OutCenter' FwdSv
      SET     M6168  ; TurnoverOutCent'FwdFault
      MPP
      ANI     Y3A6  ; Turn OutCenter' FwdSv
      SET     M6169  ; TurnoverOutCent'RevFault
1043  LD      Y0AC  ; Turn OutConv'FwdInv
      AND     B0E43  ; Auto    ModeLampT-Over
      OUT     T1583 K200  ; TurnoverOut->   FormConvTime
1049  LD      T1583  ; TurnoverOut->   FormConvTime
      SET     M6170  ; TurnoverOut->   FormConvTimeOut
; ============ Roll Forming Part ===========
1074  LDI     X72  ; Roll    ConveyorOverload
      AND     M0  ; PLC Run
      SET     M6180  ; RollFormConveyorFault
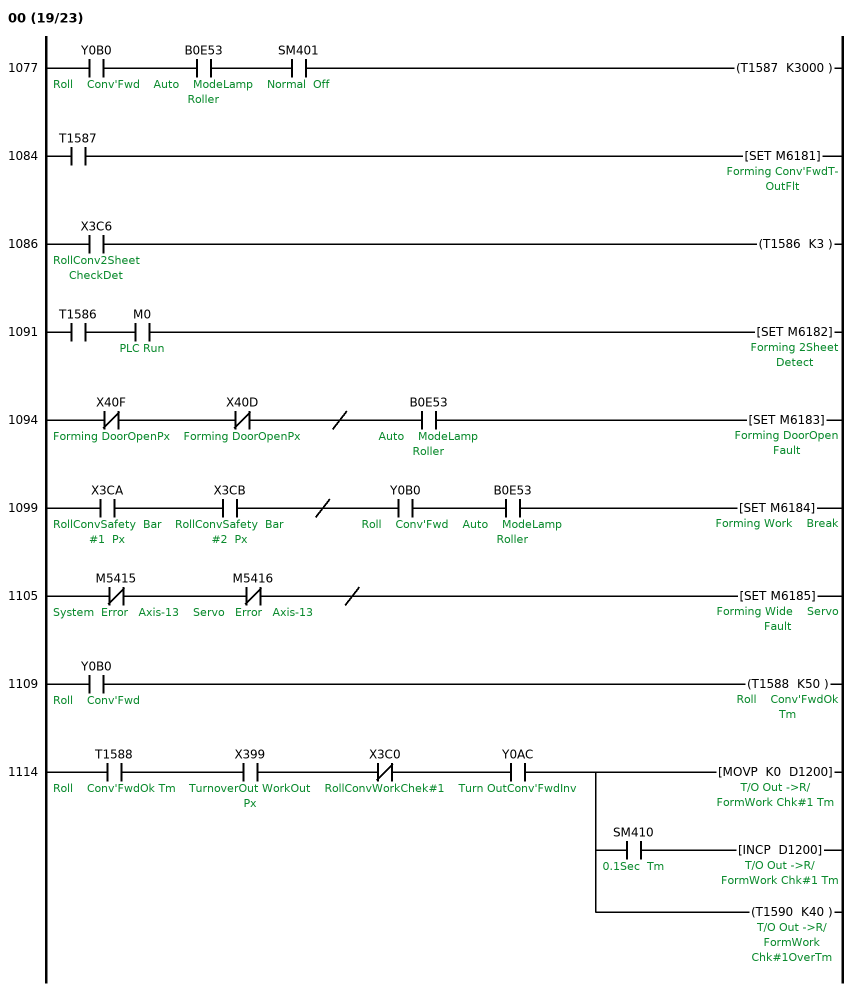
1077  LD      Y0B0  ; Roll    Conv'Fwd
      AND     B0E53  ; Auto    ModeLampRoller
      AND     SM401  ; Normal  Off
      OUT     T1587 K3000
1084  LD      T1587
      SET     M6181  ; Forming Conv'FwdT-OutFlt
1086  LD      X3C6  ; RollConv2Sheet  CheckDet
      OUT     T1586 K3
1091  LD      T1586
      AND     M0  ; PLC Run
      SET     M6182  ; Forming 2Sheet  Detect
1094  LDI     X40F  ; Forming DoorOpenPx
      ANI     X40D  ; Forming DoorOpenPx
      INV
      AND     B0E53  ; Auto    ModeLampRoller
      SET     M6183  ; Forming DoorOpenFault
1099  LD      X3CA  ; RollConvSafety  Bar #1  Px
      AND     X3CB  ; RollConvSafety  Bar #2  Px
      INV
      AND     Y0B0  ; Roll    Conv'Fwd
      AND     B0E53  ; Auto    ModeLampRoller
      SET     M6184  ; Forming Work    Break
1105  LDI     M5415  ; System  Error   Axis-13
      ANI     M5416  ; Servo   Error   Axis-13
      INV
      SET     M6185  ; Forming Wide    Servo   Fault
1109  LD      Y0B0  ; Roll    Conv'Fwd
      OUT     T1588 K50  ; Roll    Conv'FwdOk Tm
1114  LD      T1588  ; Roll    Conv'FwdOk Tm
      AND     X399  ; TurnoverOut WorkOut Px
      ANI     X3C0  ; RollConvWorkChek#1
      AND     Y0AC  ; Turn OutConv'FwdInv
      MOVP    K0 D1200  ; T/O Out ->R/FormWork Chk#1 Tm
      MPS
      AND     SM410  ; 0.1Sec  Tm
      INCP    D1200
      MPP
      OUT     T1590 K40  ; T/O Out ->R/FormWork Chk#1OverTm
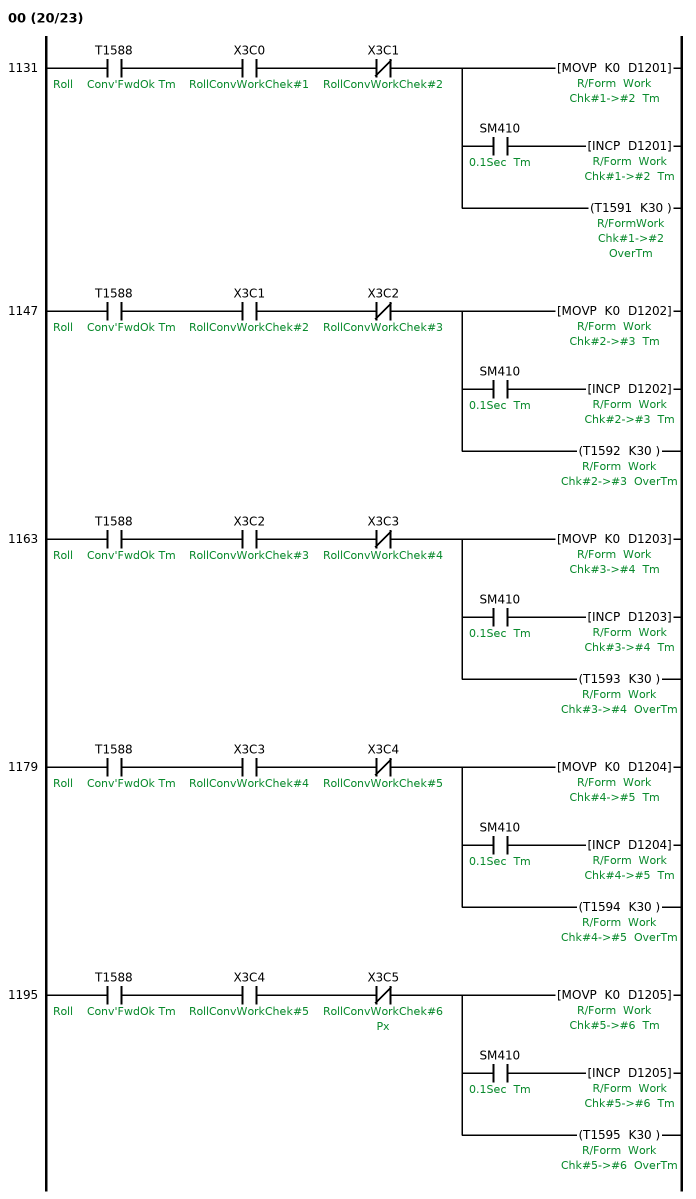
1131  LD      T1588  ; Roll    Conv'FwdOk Tm
      AND     X3C0  ; RollConvWorkChek#1
      ANI     X3C1  ; RollConvWorkChek#2
      MOVP    K0 D1201  ; R/Form  Work Chk#1->#2  Tm
      MPS
      AND     SM410  ; 0.1Sec  Tm
      INCP    D1201
      MPP
      OUT     T1591 K30  ; R/FormWork Chk#1->#2    OverTm
1147  LD      T1588  ; Roll    Conv'FwdOk Tm
      AND     X3C1  ; RollConvWorkChek#2
      ANI     X3C2  ; RollConvWorkChek#3
      MOVP    K0 D1202  ; R/Form  Work Chk#2->#3  Tm
      MPS
      AND     SM410  ; 0.1Sec  Tm
      INCP    D1202
      MPP
      OUT     T1592 K30  ; R/Form  Work Chk#2->#3  OverTm
1163  LD      T1588  ; Roll    Conv'FwdOk Tm
      AND     X3C2  ; RollConvWorkChek#3
      ANI     X3C3  ; RollConvWorkChek#4
      MOVP    K0 D1203  ; R/Form  Work Chk#3->#4  Tm
      MPS
      AND     SM410  ; 0.1Sec  Tm
      INCP    D1203
      MPP
      OUT     T1593 K30  ; R/Form  Work Chk#3->#4  OverTm
1179  LD      T1588  ; Roll    Conv'FwdOk Tm
      AND     X3C3  ; RollConvWorkChek#4
      ANI     X3C4  ; RollConvWorkChek#5
      MOVP    K0 D1204  ; R/Form  Work Chk#4->#5  Tm
      MPS
      AND     SM410  ; 0.1Sec  Tm
      INCP    D1204
      MPP
      OUT     T1594 K30  ; R/Form  Work Chk#4->#5  OverTm
1195  LD      T1588  ; Roll    Conv'FwdOk Tm
      AND     X3C4  ; RollConvWorkChek#5
      ANI     X3C5  ; RollConvWorkChek#6 Px
      MOVP    K0 D1205  ; R/Form  Work Chk#5->#6  Tm
      MPS
      AND     SM410  ; 0.1Sec  Tm
      INCP    D1205
      MPP
      OUT     T1595 K30  ; R/Form  Work Chk#5->#6  OverTm
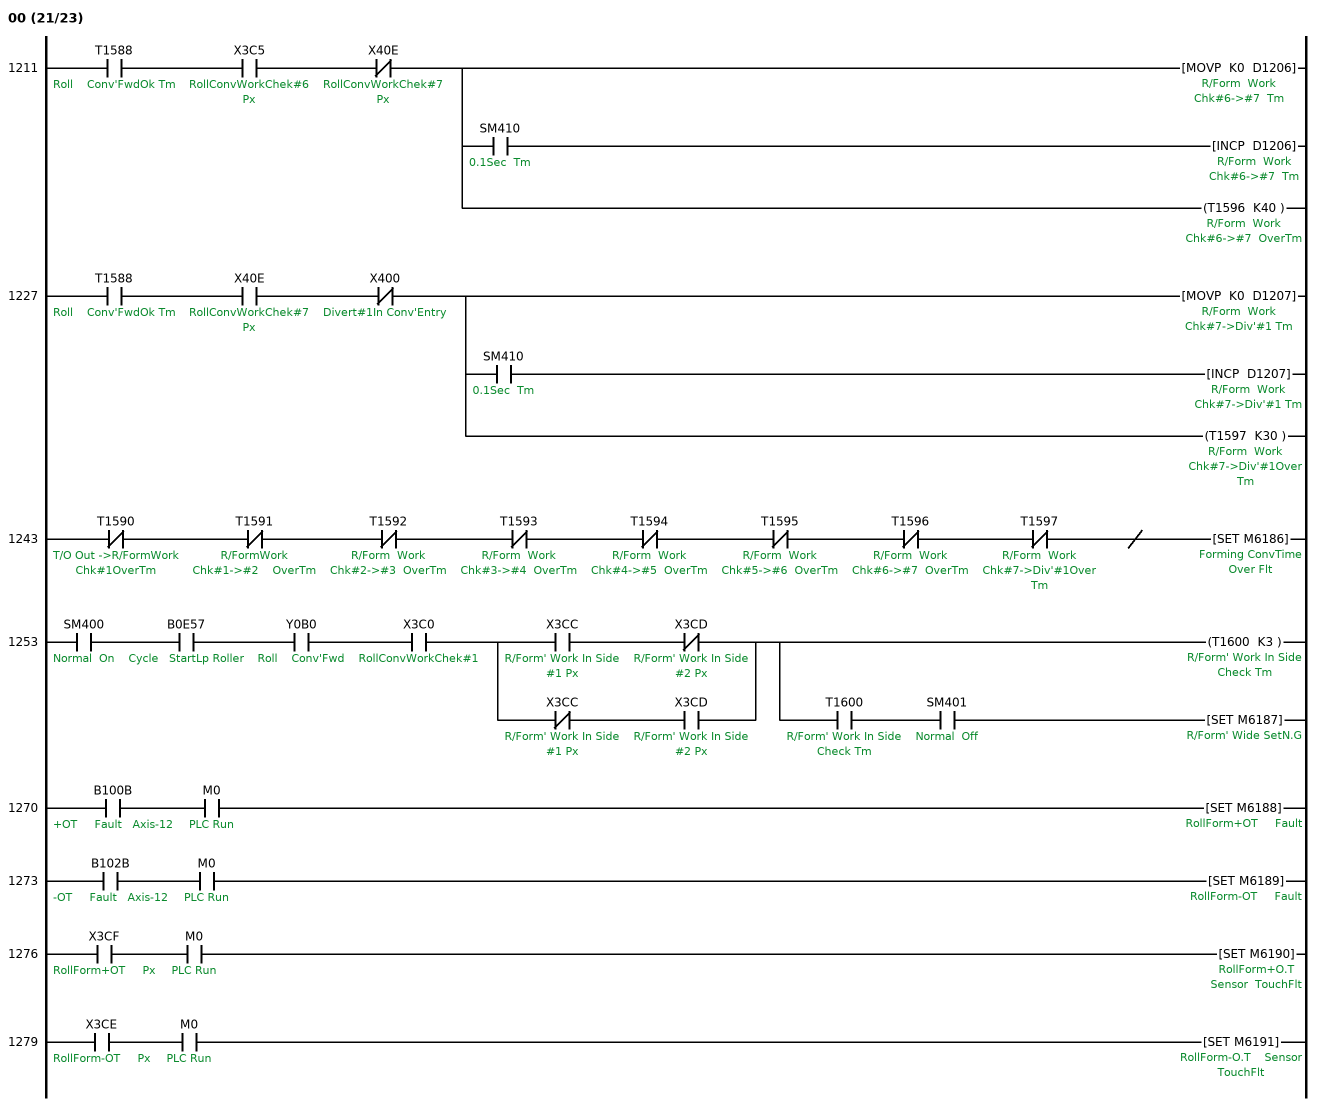
1211  LD      T1588  ; Roll    Conv'FwdOk Tm
      AND     X3C5  ; RollConvWorkChek#6 Px
      ANI     X40E  ; RollConvWorkChek#7 Px
      MOVP    K0 D1206  ; R/Form  Work Chk#6->#7  Tm
      MPS
      AND     SM410  ; 0.1Sec  Tm
      INCP    D1206
      MPP
      OUT     T1596 K40  ; R/Form  Work Chk#6->#7  OverTm
1227  LD      T1588  ; Roll    Conv'FwdOk Tm
      AND     X40E  ; RollConvWorkChek#7 Px
      ANI     X400  ; Divert#1In Conv'Entry
      MOVP    K0 D1207  ; R/Form  Work Chk#7->Div'#1 Tm
      MPS
      AND     SM410  ; 0.1Sec  Tm
      INCP    D1207
      MPP
      OUT     T1597 K30  ; R/Form  Work Chk#7->Div'#1OverTm
1243  LDI     T1590  ; T/O Out ->R/FormWork Chk#1OverTm
      ANI     T1591  ; R/FormWork Chk#1->#2    OverTm
      ANI     T1592  ; R/Form  Work Chk#2->#3  OverTm
      ANI     T1593  ; R/Form  Work Chk#3->#4  OverTm
      ANI     T1594  ; R/Form  Work Chk#4->#5  OverTm
      ANI     T1595  ; R/Form  Work Chk#5->#6  OverTm
      ANI     T1596  ; R/Form  Work Chk#6->#7  OverTm
      ANI     T1597  ; R/Form  Work Chk#7->Div'#1OverTm
      INV
      SET     M6186  ; Forming ConvTimeOver Flt
1253  LD      SM400  ; Normal  On
      AND     B0E57  ; Cycle   StartLp Roller
      AND     Y0B0  ; Roll    Conv'Fwd
      AND     X3C0  ; RollConvWorkChek#1
      LD      X3CC  ; R/Form' Work In Side #1 Px
      ANI     X3CD  ; R/Form' Work In Side #2 Px
      LDI     X3CC  ; R/Form' Work In Side #1 Px
      AND     X3CD  ; R/Form' Work In Side #2 Px
      ORB
      ANB
      OUT     T1600 K3  ; R/Form' Work In Side    Check Tm
      AND     T1600  ; R/Form' Work In Side    Check Tm
      AND     SM401  ; Normal  Off
      SET     M6187  ; R/Form' Wide SetN.G
1270  LD      B100B  ; +OT     Fault   Axis-12
      AND     M0  ; PLC Run
      SET     M6188  ; RollForm+OT     Fault
1273  LD      B102B  ; -OT     Fault   Axis-12
      AND     M0  ; PLC Run
      SET     M6189  ; RollForm-OT     Fault
1276  LD      X3CF  ; RollForm+OT     Px
      AND     M0  ; PLC Run
      SET     M6190  ; RollForm+O.T    Sensor  TouchFlt
1279  LD      X3CE  ; RollForm-OT     Px
      AND     M0  ; PLC Run
      SET     M6191  ; RollForm-O.T    Sensor  TouchFlt
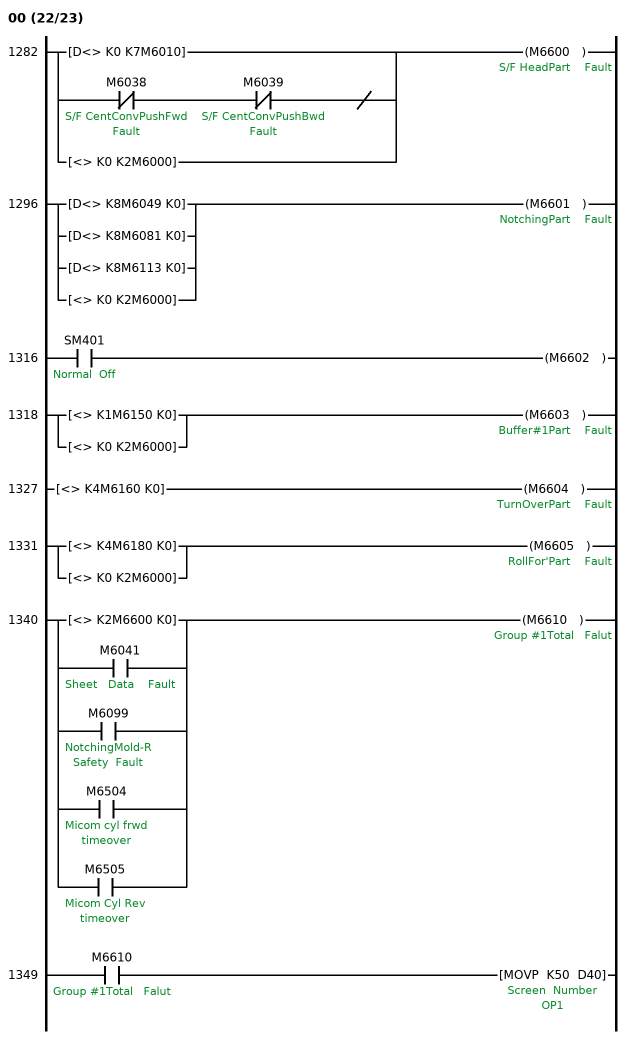
1282  LDD<>   K0 K7M6010  ; Carriage"A" OL   Fault
      LDI     M6038  ; S/F CentConvPushFwdFault
      ANI     M6039  ; S/F CentConvPushBwdFault
      INV
      ORB
      OR<>    K0 K2M6000  ; Emg-StopFault
      OUT     M6600  ; S/F HeadPart    Fault
1296  LDD<>   K8M6049 K0  ; S/F     2Sheet  Detect
      ORD<>   K8M6081 K0  ; NotchingSidePush#1FwdFlt
      ORD<>   K8M6113 K0  ; NotchingPress #5Servo   Fault
      OR<>    K0 K2M6000  ; Emg-StopFault
      OUT     M6601  ; NotchingPart    Fault
1316  LD      SM401  ; Normal  Off
      OUT     M6602
1318  LD<>    K1M6150 K0  ; Buffer#1ConveyorOverloadFault
      OR<>    K0 K2M6000  ; Emg-StopFault
      OUT     M6603  ; Buffer#1Part    Fault
1327  LD<>    K4M6160 K0  ; TurnoverInConv' Fault
      OUT     M6604  ; TurnOverPart    Fault
1331  LD<>    K4M6180 K0  ; RollFormConveyorFault
      OR<>    K0 K2M6000  ; Emg-StopFault
      OUT     M6605  ; RollFor'Part    Fault
1340  LD<>    K2M6600 K0  ; S/F HeadPart    Fault
      OR      M6041  ; Sheet   Data    Fault
      OR      M6099  ; NotchingMold-R  Safety  Fault
      OR      M6504  ; Micom cyl frwd timeover
      OR      M6505  ; Micom Cyl Rev timeover
      OUT     M6610  ; Group #1Total   Falut
1349  LD      M6610  ; Group #1Total   Falut
      MOVP    K50 D40  ; Screen  Number  OP1
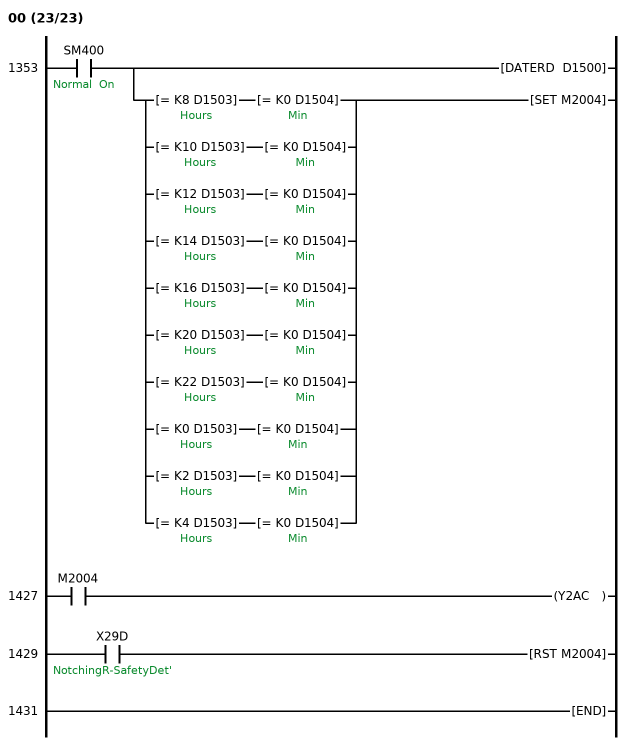
1353  LD      SM400  ; Normal  On
      DATERD  D1500
      LD=     K8 D1503  ; Hours
      AND=    K0 D1504  ; Min
      LD=     K10 D1503  ; Hours
      AND=    K0 D1504  ; Min
      ORB
      LD=     K12 D1503  ; Hours
      AND=    K0 D1504  ; Min
      ORB
      LD=     K14 D1503  ; Hours
      AND=    K0 D1504  ; Min
      ORB
      LD=     K16 D1503  ; Hours
      AND=    K0 D1504  ; Min
      ORB
      LD=     K20 D1503  ; Hours
      AND=    K0 D1504  ; Min
      ORB
      LD=     K22 D1503  ; Hours
      AND=    K0 D1504  ; Min
      ORB
      LD=     K0 D1503  ; Hours
      AND=    K0 D1504  ; Min
      ORB
      LD=     K2 D1503  ; Hours
      AND=    K0 D1504  ; Min
      ORB
      LD=     K4 D1503  ; Hours
      AND=    K0 D1504  ; Min
      ORB
      ANB
      SET     M2004
1427  LD      M2004
      OUT     Y2AC
1429  LD      X29D  ; NotchingR-SafetyDet'
      RST     M2004
1431  END
END_PROGRAM

PROGRAM 05  // Position Start
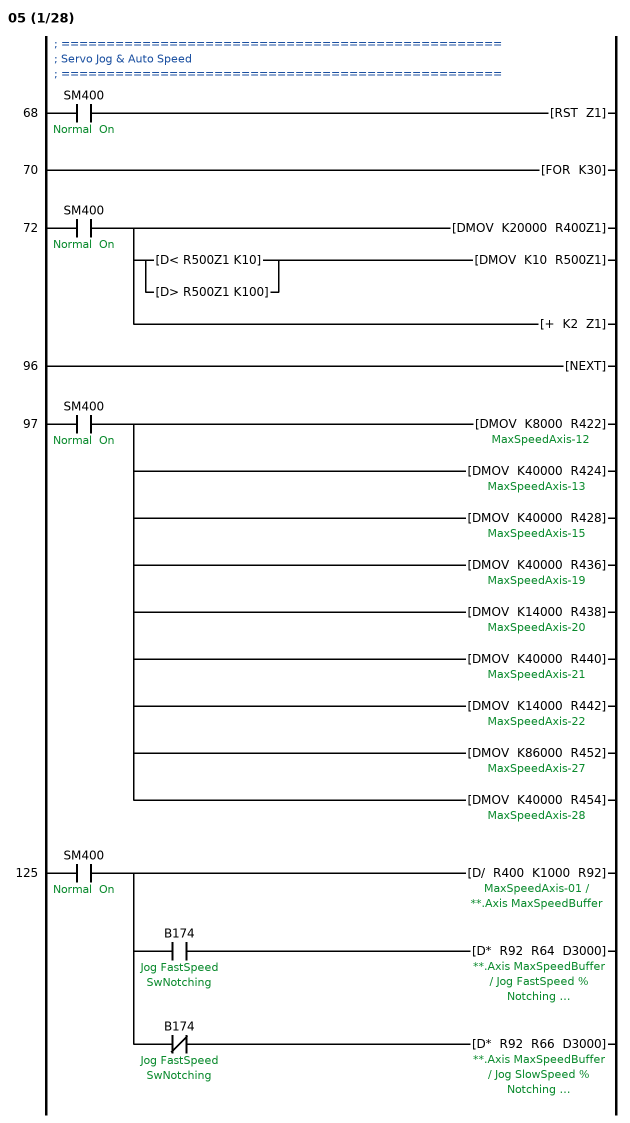
; =================================================
; Servo Jog & Auto Speed
; =================================================
68    LD      SM400  ; Normal  On
      RST     Z1
70    FOR     K30
72    LD      SM400  ; Normal  On
      DMOV    K20000 R400Z1
      MPS
      LDD<    R500Z1 K10
      ORD>    R500Z1 K100
      ANB
      DMOV    K10 R500Z1
      MPP
      +       K2 Z1
96    NEXT
97    LD      SM400  ; Normal  On
      DMOV    K8000 R422  ; MaxSpeedAxis-12
      DMOV    K40000 R424  ; MaxSpeedAxis-13
      DMOV    K40000 R428  ; MaxSpeedAxis-15
      DMOV    K40000 R436  ; MaxSpeedAxis-19
      DMOV    K14000 R438  ; MaxSpeedAxis-20
      DMOV    K40000 R440  ; MaxSpeedAxis-21
      DMOV    K14000 R442  ; MaxSpeedAxis-22
      DMOV    K86000 R452  ; MaxSpeedAxis-27
      DMOV    K40000 R454  ; MaxSpeedAxis-28
125   LD      SM400  ; Normal  On
      D/      R400 K1000 R92  ; MaxSpeedAxis-01 / **.Axis MaxSpeedBuffer
      MPS
      AND     B174  ; Jog FastSpeed SwNotching
      D*      R92 R64 D3000  ; Jog FastSpeed % Notching / JogSpeedAxis-01
      MPP
      ANI     B174  ; Jog FastSpeed SwNotching
      D*      R92 R66 D3000  ; Jog SlowSpeed % Notching
